// TIA Portal project "Playground Swing Timer" (V17)
// Playground Swing Timer
// When a child starts swinging, a timer should count down from 30 sec. An Alarm should sound when time is up.
// A reset button will start Countdown again.

(* hardware
DEVICE "S7-1200 station_1"  S7-1200 Station
   slot 0: "Rack_0"  S7-1200 Rack  Rack  V1.0
   slot 1: "PLC_1"  CPU 1215C AC/DC/Rly  6ES7 215-1BG40-0XB0  V4.5
*)

// ===== PLC "PLC_1"  CPU 1215C AC/DC/Rly =====

VAR_GLOBAL   // PLC tag table "Default tag table"
   "Swing start sensor" AT %I0.0 : Bool;
   "Reset button" AT %I0.1 : Bool;
   "Alarm" AT %Q0.0 : Bool;
   "PB" AT %I0.2 : Bool;
   "Tag_1" AT %M0.0 : Bool;
END_VAR

// folder: System blocks/Program resources

DATA_BLOCK "IEC_Timer_0_DB"   // DB1
{ S7_Optimized_Access := 'TRUE' }
AUTHOR : Simatic
FAMILY : IEC
NAME : IEC_TMR
VERSION : 1.0
// stored: InstanceOfName IEC_TIMER
"IEC_TIMER"
BEGIN
END_DATA_BLOCK

// folder: (top level)

ORGANIZATION_BLOCK "Main"   // OB1, LAD, ProgramCycle
TITLE = "Main Program Sweep (Cycle)"
{ S7_Optimized_Access := 'TRUE' }
VERSION : 0.1
   VAR_INPUT
      Initial_Call : Bool;   // Initial call of this OB
      Remanence : Bool;   // =True, if remanent data are available
   END_VAR
BEGIN

REGION Network 1
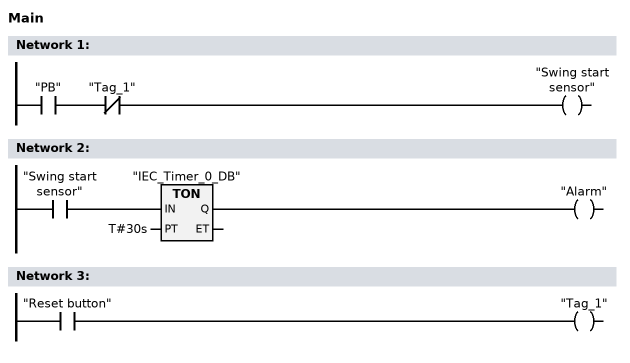
   RUNG wire#powerrail
      Contact( "PB" )
      I_Contact( "Tag_1" )
      Coil( "Swing start sensor" )
   END_RUNG
   // the same network as SCL:
   "Swing start sensor" := "PB" AND NOT "Tag_1";
END_REGION

REGION Network 2
   "IEC_Timer_0_DB".TON(IN := "Swing start sensor", PT := T#30s);
   "Alarm" := "IEC_Timer_0_DB".Q;
END_REGION

REGION Network 3
   RUNG wire#powerrail
      Contact( "Reset button" )
      Coil( "Tag_1" )
   END_RUNG
   // the same network as SCL:
   "Tag_1" := "Reset button";
END_REGION
END_ORGANIZATION_BLOCK